// TIA Portal V14 export
ORGANIZATION_BLOCK "Startup"   // OB100, SCL
// stored: AutoNumber true
BEGIN
END_ORGANIZATION_BLOCK
